(* IEC 61131-3 sources: mect_apps/TP1043_CAN/CANopenClient_PLC, 8 files *)

(* ---- CANopenClient_CAN.gvl ---- *)
(* Global var file *)
VAR_GLOBAL
	ch1_CAN1_IN_DIG_8_1 AT %IB3.4096: BYTE;
	ch1_CAN1_IN_DIG_8_1_1 AT %IX3.4096.0: BOOL;
	ch1_CAN1_IN_DIG_8_1_2 AT %IX3.4096.1: BOOL;
	ch1_CAN1_IN_DIG_8_1_3 AT %IX3.4096.2: BOOL;
	ch1_CAN1_IN_DIG_8_1_4 AT %IX3.4096.3: BOOL;
	ch1_CAN1_IN_DIG_8_1_5 AT %IX3.4096.4: BOOL;
	ch1_CAN1_IN_DIG_8_1_6 AT %IX3.4096.5: BOOL;
	ch1_CAN1_IN_DIG_8_1_7 AT %IX3.4096.6: BOOL;
	ch1_CAN1_IN_DIG_8_1_8 AT %IX3.4096.7: BOOL;

	ch1_CAN1_IN_DIG_8_2 AT %IB3.4097: BYTE;

	ch1_CAN1_OUT_DIG_8_1 AT %QB3.4096: BYTE;
	ch1_CAN1_OUT_DIG_8_1_1 AT %QX3.4096.0: BOOL;
	ch1_CAN1_OUT_DIG_8_1_2 AT %QX3.4096.1: BOOL;
	ch1_CAN1_OUT_DIG_8_1_3 AT %QX3.4096.2: BOOL;
	ch1_CAN1_OUT_DIG_8_1_4 AT %QX3.4096.3: BOOL;
	ch1_CAN1_OUT_DIG_8_1_5 AT %QX3.4096.4: BOOL;
	ch1_CAN1_OUT_DIG_8_1_6 AT %QX3.4096.5: BOOL;
	ch1_CAN1_OUT_DIG_8_1_7 AT %QX3.4096.6: BOOL;
	ch1_CAN1_OUT_DIG_8_1_8 AT %QX3.4096.7: BOOL;

	ch1_CAN1_OUT_DIG_8_2 AT %QB3.4097: BYTE;
	ch1_CAN1_IN_AN_1 AT %IW3.8192: INT;
	ch1_CAN1_IN_AN_2 AT %IW3.8194: INT;
	ch1_3 AT %IW3.8196: INT;
	ch1_4 AT %IW3.8198: INT;
	ch1_5 AT %IW3.8200: INT;
	ch1_6 AT %IW3.8202: INT;
	ch1_CAN1_OUT_AN_1 AT %QW3.8192: INT;
	PLC_CAN1_IN_DIG_8_1 AT %MB0.5380: BYTE;
	PLC_CAN1_IN_DIG_8_2 AT %MB0.5384: BYTE;
	PLC_CAN1_OUT_DIG_8_1 AT %MB0.5388: BYTE;
	PLC_CAN1_OUT_DIG_8_2 AT %MB0.5392: BYTE;
	PLC_CAN1_IN_AN_1 AT %MW0.5396: INT;
	PLC_CAN1_IN_AN_2 AT %MW0.5400: INT;
	PLC_3 AT %MW0.5404: INT;
	PLC_4 AT %MW0.5408: INT;
	PLC_5 AT %MW0.5412: INT;
	PLC_6 AT %MW0.5416: INT;
	PLC_CAN1_OUT_AN_1 AT %MW0.5420: INT;
END_VAR

(* ---- Resource1.gvl ---- *)
(* Global variable file *)
VAR_GLOBAL
DigitalInput_3 AT %MW0.5380:UINT;
DigitalInput_4 AT %MW0.5384:UINT;
DigitalOutput_1 AT %MW0.5388:UINT;
DigitalOutput_2 AT %MW0.5392:UINT;
AnalogInput_1 AT %MW0.5396:INT;
AnalogInput_2 AT %MW0.5400:INT;
END_VAR

(* ---- fb_HW119_AlarmsMngr.st ---- *)
(*[[
]]*)
FUNCTION_BLOCK fb_HW119_AlarmsMngr
#import "Resource1.gvl"
#import "crosstable.gvl"
VAR_INPUT
END_VAR
VAR
	Index:DINT;			(* indice di scansione della CT degli allarmi	*)
	SourceAddr:INT;		(* indirizzo della variabile sorgente	*)
	CompareAdddr:INT;	(* indirizzo della variabile di confronto	*)
	CompareVal:DWORD;	(* valore di confronto	*)
	TagAddr:INT;		(* indirizzo della variabile di allarme	*)
	ERRFlag:BOOL;		(* flag d segnalazione errore nell'esecuzioe di una funzione	*)
	ERRORVAL:DWORD:=16#00000001;	(* *)
	tmp:DWORD;			(* variabile di appoggio	*)
	tmpOld:DWORD;		(* variabile di appoggio	*)
END_VAR
(*
	Blocco funzione per la gestione degli alalrmi/eventi

*)

	IF Index < DimAlarmsCT AND ALCrossTable[Index].ALTag <> '' THEN
		SourceAddr:=WORD_TO_INT(HW119_GetAddr(ALCrossTable[Index].ALSource));		(* ricava l'indirizzo della varibile sorgente*)
		IF SourceAddr = WORD_TO_INT(16#FFFF)  OR SourceAddr > DINT_TO_INT(DimCrossTable) OR SourceAddr = 0  THEN									(* controlla il risultato della funzione*)
			ERRFlag:=TRUE;
		ELSE
			IF	CrossTable[SourceAddr].Error > 0 AND CrossTable[SourceAddr].Protocol<>100 THEN			(* verifica che il valore sia stato aggiornato	*)
				ERRFlag:=TRUE;
			ELSE
				CompareAdddr:=-1;
				IF ALCrossTable[Index].ALCompareVar = '' THEN
					CompareVal:=ALCrossTable[Index].ALCompareVaL;					(* variabile di confronto nulla -> rileva il valore di confronto*)
				ELSE
					CompareAdddr:=WORD_TO_INT(HW119_GetAddr(ALCrossTable[Index].ALCompareVar));	(* ricava l'indirizzo della varibile di confronto *)

					IF CompareAdddr = WORD_TO_INT(16#FFFF) OR CompareAdddr > DINT_TO_INT(DimCrossTable) OR CompareAdddr = 0 THEN					(* controlla se la variable di controllo corretta*)
						ERRFlag:=TRUE;
					ELSE
						IF CrossTable[CompareAdddr].Error > 0 AND CrossTable[CompareAdddr].Protocol<>100 THEN	(* verifica  se la variabile di controllo è nella CT*)
							ERRFlag:=TRUE;
						ELSE
							CompareVal:=ARRAY_CROSSTABLE_INPUT[CompareAdddr];
						END_IF;
					END_IF;
				END_IF;
				TagAddr:=WORD_TO_INT(HW119_GetAddr(ALCrossTable[Index].ALTag));		(* ricavo l'indirizzo della varibile destinazione*)
				IF TagAddr = WORD_TO_INT(16#FFFF) OR TagAddr > DINT_TO_INT(DimCrossTable) OR TagAddr = 0 THEN
					ERRFlag:=TRUE;
				END_IF;
			END_IF;
		END_IF;

		IF NOT ERRFlag	THEN						(* Se i valori letti da CT sono corenti effettua il check di allarme	*)
			tmp:=UINT_TO_DWORD(ALCrossTable[Index].ALOperator)	AND 16#FF00	;	(* controlla l'operazione da eseguire *)
			CASE DWORD_TO_INT(tmp) OF
(*  operatore >	*)		16#100 :
							IF ARRAY_CROSSTABLE_INPUT[SourceAddr] > CompareVal	 THEN
								IF  ALCrossTable[Index].ALFilterCount=0  THEN
									ARRAY_CROSSTABLE_INPUT[TagAddr]:=ERRORVAL;
								ELSE
									ALCrossTable[Index].ALFilterCount:=ALCrossTable[Index].ALFilterCount-1;
								END_IF;
							ELSE
								ARRAY_CROSSTABLE_INPUT[TagAddr]:=0;
								ALCrossTable[Index].ALFilterCount:=ALCrossTable[Index].ALFilterTime;
							END_IF;
(*  operatore >=	*)	16#200 :
							IF ARRAY_CROSSTABLE_INPUT[SourceAddr] >= CompareVal	 THEN
								IF  ALCrossTable[Index].ALFilterCount=0  THEN
									ARRAY_CROSSTABLE_INPUT[TagAddr]:=ERRORVAL;
								ELSE
									ALCrossTable[Index].ALFilterCount:=ALCrossTable[Index].ALFilterCount-1;
								END_IF;
							ELSE
								ARRAY_CROSSTABLE_INPUT[TagAddr]:=0;

							END_IF;
(*  operatore <	*)		16#300 :
							IF ARRAY_CROSSTABLE_INPUT[SourceAddr] < CompareVal	 THEN
								IF  ALCrossTable[Index].ALFilterCount=0  THEN
									ARRAY_CROSSTABLE_INPUT[TagAddr]:=ERRORVAL;

								ELSE
									ALCrossTable[Index].ALFilterCount:=ALCrossTable[Index].ALFilterCount-1;
								END_IF;
							ELSE
								ARRAY_CROSSTABLE_INPUT[TagAddr]:=0;
								ALCrossTable[Index].ALFilterCount:=ALCrossTable[Index].ALFilterTime;
							END_IF;
(*  operatore <=	*)	16#400 :
							IF ARRAY_CROSSTABLE_INPUT[SourceAddr] <= CompareVal	 THEN
								IF  ALCrossTable[Index].ALFilterCount=0  THEN
									ARRAY_CROSSTABLE_INPUT[TagAddr]:=ERRORVAL;

								ELSE
									ALCrossTable[Index].ALFilterCount:=ALCrossTable[Index].ALFilterCount-1;
								END_IF;
							ELSE
								ARRAY_CROSSTABLE_INPUT[TagAddr]:=0;
								ALCrossTable[Index].ALFilterCount:=ALCrossTable[Index].ALFilterTime;
							END_IF;
(*  operatore =	*)		16#500 :
							IF ARRAY_CROSSTABLE_INPUT[SourceAddr] = CompareVal	 THEN
								IF  ALCrossTable[Index].ALFilterCount=0  THEN
									ARRAY_CROSSTABLE_INPUT[TagAddr]:=ERRORVAL;

								ELSE
									ALCrossTable[Index].ALFilterCount:=ALCrossTable[Index].ALFilterCount-1;
								END_IF;
							ELSE
								ARRAY_CROSSTABLE_INPUT[TagAddr]:=0;
								ALCrossTable[Index].ALFilterCount:=ALCrossTable[Index].ALFilterTime;
							END_IF;
(*  operatore <>	*)	16#600 :
							IF ARRAY_CROSSTABLE_INPUT[SourceAddr] <> CompareVal	 THEN
								IF  ALCrossTable[Index].ALFilterCount=0  THEN
									ARRAY_CROSSTABLE_INPUT[TagAddr]:=ERRORVAL;

								ELSE
									ALCrossTable[Index].ALFilterCount:=ALCrossTable[Index].ALFilterCount-1;
								END_IF;
							ELSE
								ARRAY_CROSSTABLE_INPUT[TagAddr]:=0;
								ALCrossTable[Index].ALFilterCount:=ALCrossTable[Index].ALFilterTime;
							END_IF;

						ELSE
(*controllo a bit *)

							tmp:= SHR(ARRAY_CROSSTABLE_INPUT[SourceAddr], WORD_TO_INT ( UINT_TO_WORD ( ALCrossTable[Index].ALOperator) AND 16#00FF)-1 );
							tmp:=tmp AND 16#1;
							(*controllo a bit sui livelli*)

							IF CompareAdddr = -1 THEN

								IF tmp = CompareVal	THEN
									IF  ALCrossTable[Index].ALFilterCount=0  THEN
										ARRAY_CROSSTABLE_INPUT[TagAddr]:=ERRORVAL;

									ELSE
										ALCrossTable[Index].ALFilterCount:=ALCrossTable[Index].ALFilterCount-1;
									END_IF;
								ELSE
									ARRAY_CROSSTABLE_INPUT[TagAddr]:=0;
									ALCrossTable[Index].ALFilterCount:=ALCrossTable[Index].ALFilterTime;
								END_IF;
(* controllo  transizioni*)
							ELSIF CompareAdddr=SourceAddr 	THEN
(* allarme su fronte di salita*)
								tmpOld:= SHR(CrossTable[SourceAddr].OldVal, WORD_TO_INT ( UINT_TO_WORD ( ALCrossTable[Index].ALOperator) AND 16#00FF)-1 );
								tmpOld:=tmpOld AND 16#1;
								IF		tmp = 16#01 AND 	tmpOld=16#00 AND ALCrossTable[Index].ALCompareVal =  FRONTE_SALITA	THEN
								 	ARRAY_CROSSTABLE_INPUT[TagAddr]:=ERRORVAL;
(* allarme su fronte di discesa*)
								ELSIF	tmp = 16#00  AND 	tmpOld=16#01 AND ALCrossTable[Index].ALCompareVal =  FRONTE_DISCESA	THEN
								 	ARRAY_CROSSTABLE_INPUT[TagAddr]:=ERRORVAL;
								ELSIF ALCrossTable[Index].ALCompareVal =  FRONTE_SALITA AND tmp=16#00 THEN
									ARRAY_CROSSTABLE_INPUT[TagAddr]:=0;
								ELSIF ALCrossTable[Index].ALCompareVal =  FRONTE_DISCESA AND tmp= 16#01 THEN
									ARRAY_CROSSTABLE_INPUT[TagAddr]:=0;
								END_IF;
								IF tmp = 0 THEN
									tmp:=16#FFFFFFFE;
									CrossTable[SourceAddr].OldVal:=CrossTable[SourceAddr].OldVal AND ROL(tmp, WORD_TO_INT ( UINT_TO_WORD ( ALCrossTable[Index].ALOperator) AND 16#00FF)-1 );
								ELSE
									CrossTable[SourceAddr].OldVal:=CrossTable[SourceAddr].OldVal OR ROL(tmp, WORD_TO_INT ( UINT_TO_WORD ( ALCrossTable[Index].ALOperator) AND 16#00FF)-1 );
								END_IF;
							END_IF;

			END_CASE;
		END_IF;
		Index:=Index+1;
		ERRFlag:=FALSE;
	ELSE
		Index:=1;
	END_IF;

END_FUNCTION_BLOCK

(* ---- fb_HW119_MODBUS.st ---- *)
(*[[
]]*)
FUNCTION_BLOCK fb_HW119_MODBUS
#import "Resource1.gvl"
#import "crosstable.gvl"
VAR_INPUT
	RdWr:WORD;
	address:INT;
	Index:int;
	Protocol:STRING;
END_VAR
VAR_OUTPUT
	Error:UINT;
END_VAR
VAR
	FunctRes:UINT;
	HeadAddr:INT;
	I:INT;
	STEPS:INT;
	RW:WORD;
	COUNT_ERR:UDINT:=0;
	addr:INT;
	COUNT_CICLI:UDINT;
	regs:INT;
	LowByte:BYTE;
	BOOL_Data:	ARRAY[0..259]	OF BYTE;
	INT_Data:	ARRAY[0..259]	OF UINT;
	tempo1:TIME;
	tempo2:TIME;
	Index_A:int;
	tmpARRAY_CROSSTABLE_OUTPUT:	ARRAY[0..19] OF DWORD;
END_VAR

	tempo1:=TIM_Get();
(*	TRIGGER02:=1;
	TRIGGER01:=1;
	*)

		RW:=RdWr;
		HeadAddr:=address;
		addr:=address;
		Index_A:=Index;

		IF RW > 0   THEN											(* Variabile abilitata*)

			COUNT_CICLI:=COUNT_CICLI+1;
			FunctRes:= MODBUS_SET_SLAVE(Protocol,CrossTable[HeadAddr].NodeId);
			IF FunctRes = 0  THEN										(* Funzione andata a buon fine*)
				MODBUS_ERR[10]:=2;
				IF RW = READ	THEN									(* OPERAZIONE DI LETTURA	*)
					TRIGGER02:=1;
					regs:=0;
					IF Index_A > 0 THEN
						ARRAY_QUEUE_OUTPUT[Index_A]:=STATO_BUSY_READ;	(* metto busy read l'intero blocco*)
					END_IF;
					FOR I:=0 TO CrossTable[HeadAddr].NReg-1 DO				(*  calcolo del numero di letture modbus da effettuare*)

						CASE CrossTable[HeadAddr+I].Types OF
							FLOATABCD,UDINTABCD,DINTABCD:		regs:=regs+2;
							FLOATDCBA,UDINTDCBA,DINTDCBA:		regs:=regs+2;
							FLOATCDAB,UDINTCDAB,DINTCDAB:		regs:=regs+2;
							FLOATBADC,UDINTBADC,DINTBADC:		regs:=regs+2;
						ELSE
							regs:=regs+1;
						END_CASE;
				   	END_FOR;
					IF CrossTable[HeadAddr].Types = BIT THEN			(* richiesta di lettura a bit	*)
						FunctRes:=  MODBUS_READ_BITS (Protocol,CrossTable[HeadAddr].Address,INT_TO_UINT(regs),BOOL_Data);
					ELSE
						FunctRes:= MODBUS_READ_REGISTERS (Protocol,CrossTable[HeadAddr].Address,INT_TO_UINT(regs),INT_Data);
					END_IF;
					IF FunctRes = 0  THEN								(* Funzione andata a buon fine*)
						Error:=0;
						MODBUS_ERR[11]:=2;
						ErrorsState:=ErrorsState AND 16#FF7F;
						CrossTable[HeadAddr].Error:=0;						(* segnala valore valido	*)
						I:=0;
						REPEAT
							CASE CrossTable[HeadAddr].Types OF
								FLOATABCD,UDINTABCD,DINTABCD :		STEPS:=2;
								FLOATDCBA,UDINTDCBA,DINTDCBA:		STEPS:=2;
								FLOATCDAB,UDINTCDAB,DINTCDAB:		STEPS:=2;
								FLOATBADC,UDINTBADC,DINTBADC:		STEPS:=2;
							ELSE
								STEPS:=1;
							END_CASE;
							CASE CrossTable[addr].Types	OF				(* in funzione del tipo di dato sistema la variabile	*)
								FLOATABCD,UDINTABCD,DINTABCD:
									ARRAY_CROSSTABLE_INPUT[addr]:=0;
									ARRAY_CROSSTABLE_INPUT[addr]:=UINT_TO_DWORD(INT_Data[I]) OR SHL(UINT_TO_DWORD(INT_Data[I+1]),16) ;
							(*		DummyFloat:=DWORD_TO_REAL(ARRAY_CROSSTABLE_INPUT[addr+I]);*)

								FLOATDCBA,UDINTDCBA,DINTDCBA:
									ARRAY_CROSSTABLE_INPUT[addr]:=0;
									LowByte:=UINT_TO_BYTE(INT_Data[I]);
									INT_Data[I]:= WORD_TO_UINT(SHR(UINT_TO_WORD(INT_Data[I]),8));
									INT_Data[I]:=	WORD_TO_UINT(UINT_TO_WORD(INT_Data[I]) OR  SHL(BYTE_TO_WORD(LowByte),8));
									LowByte:=UINT_TO_BYTE(INT_Data[I+1]);
									INT_Data[I+1]:= WORD_TO_UINT(SHR(UINT_TO_WORD(INT_Data[I+1]),8));
									INT_Data[I+1]:=	WORD_TO_UINT(UINT_TO_WORD(INT_Data[I+1]) OR  SHL(BYTE_TO_WORD(LowByte),8));
									ARRAY_CROSSTABLE_INPUT[addr]:=UINT_TO_DWORD(INT_Data[I+1]) OR SHL(UINT_TO_DWORD(INT_Data[I]),16) ;

								FLOATCDAB,UDINTCDAB,DINTCDAB:
									ARRAY_CROSSTABLE_INPUT[addr]:=0;
									ARRAY_CROSSTABLE_INPUT[addr]:=UINT_TO_DWORD(INT_Data[I+1]) OR SHL(UINT_TO_DWORD(INT_Data[I]),16) ;

								FLOATBADC,UDINTBADC,DINTBADC:
									ARRAY_CROSSTABLE_INPUT[addr]:=0;
									LowByte:=UINT_TO_BYTE(INT_Data[I]);
									INT_Data[I]:= WORD_TO_UINT(SHR(UINT_TO_WORD(INT_Data[I]),8));
									INT_Data[I]:=	WORD_TO_UINT(UINT_TO_WORD(INT_Data[I]) OR  SHL(BYTE_TO_WORD(LowByte),8));
									LowByte:=UINT_TO_BYTE(INT_Data[I+1]);
									INT_Data[I+1]:= WORD_TO_UINT(SHR(UINT_TO_WORD(INT_Data[I+1]),8));
									INT_Data[I+1]:=	WORD_TO_UINT(UINT_TO_WORD(INT_Data[I+1]) OR  SHL(BYTE_TO_WORD(LowByte),8));
									ARRAY_CROSSTABLE_INPUT[addr]:=UINT_TO_DWORD(INT_Data[I]) OR SHL(UINT_TO_DWORD(INT_Data[I+1]),16) ;
								UINT16:
									ARRAY_CROSSTABLE_INPUT[addr]:=UINT_TO_DWORD(INT_Data[I]);
								INT16:
									ARRAY_CROSSTABLE_INPUT[addr]:=UINT_TO_DWORD(INT_Data[I]);
								BIT:
									ARRAY_CROSSTABLE_INPUT[addr]:=BYTE_TO_DWORD(BOOL_Data[I]);
							ELSE
								ARRAY_CROSSTABLE_INPUT[addr]:=UINT_TO_DWORD(INT_Data[I]);
							END_CASE;
							addr:=addr+1;							(* punta alla successiva variabile della crosstable*)
							I:=I+STEPS;
						UNTIL I >= regs
						END_REPEAT;
						FOR I:=0 TO CrossTable[HeadAddr].NReg-1	DO
							ARRAY_STATES[HeadAddr+I]:=STATO_OK;				(* segnala lo stato della comunicazione a OK		*)
							CrossTable[HeadAddr+I].Error:=0;						(* segnala valore valido	*)
						END_FOR;
					ELSIF FunctRes > 0	THEN						(*	segnala lo stato della comunicazione a  ERR		*)
						MODBUS_ERR[11]:=3;
						ErrorsState:=ErrorsState OR 16#0080;
						Error:=FunctRes;
						FOR I:=0 TO CrossTable[HeadAddr].NReg-1	DO
							ARRAY_STATES[HeadAddr+I]:=STATO_ERR;
							CrossTable[HeadAddr+I].Error:=1;					(* segnala valore non valido *)
						END_FOR;
						COUNT_ERR:=COUNT_ERR+1;
					END_IF;
				ELSIF  RW =  WRITE_SINGLE OR RW = WRITE_MULTIPLE OR RW = WRITE_RIC_SINGLE  OR RW = WRITE_RIC_MULTIPLE    THEN												(*	OPERAZIONE DI SCRITTURA	*)
					regs:=0;
					RW:=RW AND 16#B000;
					IF RW=WRITE_SINGLE THEN							(* scrittura singola ingnoro il contenuto di Nreg*)
						IF Index_A > 0 THEN
							ARRAY_QUEUE_OUTPUT[Index_A]:=STATO_BUSY_WRITE;
							tmpARRAY_CROSSTABLE_OUTPUT[0]:=ARRAY_CROSSTABLE_OUTPUT[HeadAddr];
						ELSE
							tmpARRAY_CROSSTABLE_OUTPUT[0]:=CrossTable[HeadAddr].PLCWriteVal;
						END_IF;
						ARRAY_STATES[HeadAddr]:=STATO_RUN;
						CASE CrossTable[HeadAddr].Types OF
							FLOATABCD,UDINTABCD,DINTABCD:		regs:=2;
							FLOATDCBA,UDINTDCBA,DINTDCBA:		regs:=2;
							FLOATCDAB,UDINTCDAB,DINTCDAB:		regs:=2;
							FLOATBADC,UDINTBADC,DINTBADC:		regs:=2;
						ELSE
							regs:=1;
						END_CASE;

					ELSIF RW = WRITE_MULTIPLE THEN
						IF Index_A > 0 THEN
							ARRAY_QUEUE_OUTPUT[Index_A]:=STATO_BUSY_WRITE;
						END_IF;

						FOR I:=0 TO CrossTable[HeadAddr].NReg-1 DO				(*  calcolo del numero di letture modbus da effettuare*)
							IF Index_A > 0 THEN
								tmpARRAY_CROSSTABLE_OUTPUT[I]:=ARRAY_CROSSTABLE_OUTPUT[HeadAddr+I];
							ELSE
								tmpARRAY_CROSSTABLE_OUTPUT[I]:=CrossTable[HeadAddr+I].PLCWriteVal;
							END_IF;

							ARRAY_STATES[HeadAddr+I]:=STATO_RUN;
							CASE CrossTable[HeadAddr+I].Types OF
								FLOATABCD,UDINTABCD,DINTABCD:		regs:=regs+2;
								FLOATDCBA,UDINTDCBA,DINTDCBA:		regs:=regs+2;
								FLOATCDAB,UDINTCDAB,DINTCDAB:		regs:=regs+2;
								FLOATBADC,UDINTBADC,DINTBADC:		regs:=regs+2;
							ELSE
								regs:=regs+1;
							END_CASE;
					   	END_FOR;
					END_IF;

					I:=0;
					REPEAT
						CASE CrossTable[addr].Types OF
							FLOATABCD,UDINTABCD,DINTABCD :		STEPS:=2;
							FLOATDCBA,UDINTDCBA,DINTDCBA:		STEPS:=2;
							FLOATCDAB,UDINTCDAB,DINTCDAB:		STEPS:=2;
							FLOATBADC,UDINTBADC,DINTBADC:		STEPS:=2;
						ELSE
							STEPS:=1;
						END_CASE;

						CASE CrossTable[addr].Types	OF				(* in funzione del tipo di dato arrangia la variabile	*)

							FLOATDCBA,UDINTDCBA,DINTDCBA:
								INT_Data[I+1]:=DWORD_TO_UINT(tmpARRAY_CROSSTABLE_OUTPUT[addr-HeadAddr] AND 16#0000FFFF);
								INT_Data[I]:=DWORD_TO_UINT(SHR(tmpARRAY_CROSSTABLE_OUTPUT[addr-HeadAddr],16) AND 16#0000FFFF);
								LowByte:=UINT_TO_BYTE(INT_Data[I]);
								INT_Data[I]:= WORD_TO_UINT(SHR(UINT_TO_WORD(INT_Data[I]),8));
								INT_Data[I]:=	WORD_TO_UINT(UINT_TO_WORD(INT_Data[I]) OR  SHL(BYTE_TO_WORD(LowByte),8));
								LowByte:=UINT_TO_BYTE(INT_Data[I+1]);
								INT_Data[I+1]:= WORD_TO_UINT(SHL(UINT_TO_WORD(INT_Data[I+1]),8));
								INT_Data[I+1]:=	WORD_TO_UINT(UINT_TO_WORD(INT_Data[I+1]) OR  SHL(BYTE_TO_WORD(LowByte),8));

							FLOATCDAB,UDINTCDAB,DINTCDAB:
								INT_Data[I+1]:=DWORD_TO_UINT(tmpARRAY_CROSSTABLE_OUTPUT[addr-HeadAddr] AND 16#0000FFFF);
								INT_Data[I]:=DWORD_TO_UINT(SHL(tmpARRAY_CROSSTABLE_OUTPUT[addr-HeadAddr],16) AND 16#0000FFFF);

							FLOATBADC,UDINTBADC,DINTBADC:
								INT_Data[I]:=DWORD_TO_UINT(tmpARRAY_CROSSTABLE_OUTPUT[addr-HeadAddr] AND 16#0000FFFF);
								INT_Data[I+1]:=DWORD_TO_UINT(SHR(tmpARRAY_CROSSTABLE_OUTPUT[addr-HeadAddr],16) AND 16#0000FFFF);
								LowByte:=UINT_TO_BYTE(INT_Data[I]);
								INT_Data[I]:= WORD_TO_UINT(SHR(UINT_TO_WORD(INT_Data[I]),8));
								INT_Data[I]:=	WORD_TO_UINT(UINT_TO_WORD(INT_Data[I]) OR  SHL(BYTE_TO_WORD(LowByte),8));
								LowByte:=UINT_TO_BYTE(INT_Data[I+1]);
								INT_Data[I+1]:= WORD_TO_UINT(SHL(UINT_TO_WORD(INT_Data[I+1]),8));
								INT_Data[I+1]:=	WORD_TO_UINT(UINT_TO_WORD(INT_Data[I+1]) OR  SHL(BYTE_TO_WORD(LowByte),8));

							UINT16:	INT_Data[I]:=DWORD_TO_UINT(tmpARRAY_CROSSTABLE_OUTPUT[addr-HeadAddr] AND 16#0000FFFF);

							INT16:	INT_Data[I]:=DWORD_TO_UINT(tmpARRAY_CROSSTABLE_OUTPUT[addr-HeadAddr] AND 16#0000FFFF);

							BIT:	BOOL_Data[I]:=DWORD_TO_BYTE(tmpARRAY_CROSSTABLE_OUTPUT[addr-HeadAddr] AND 16#0000FFFF);

						ELSE
							INT_Data[I]:=DWORD_TO_UINT(tmpARRAY_CROSSTABLE_OUTPUT[addr-HeadAddr] AND 16#0000FFFF);
							INT_Data[I+1]:=DWORD_TO_UINT(SHR(tmpARRAY_CROSSTABLE_OUTPUT[addr-HeadAddr],16) AND 16#0000FFFF);

						END_CASE;
						I:=I+STEPS;
						addr:=addr+1;							(* punta alla successiva variabile della crosstable*)

					UNTIL I >= regs
				    END_REPEAT;

					IF  CrossTable[HeadAddr].Types = BIT	THEN		(* richiesta scrittura a bit*)
						FunctRes:= MODBUS_WRITE_BITS (Protocol,CrossTable[HeadAddr].Address,INT_TO_UINT(regs),BOOL_Data);
					ELSE												(*riciesta scrittura a word*)
						IF regs = 1	THEN
							FunctRes:= MODBUS_WRITE_REGISTER (Protocol,CrossTable[HeadAddr].Address,INT_Data[0]);
						ELSE
							FunctRes:= MODBUS_WRITE_REGISTERS (Protocol,CrossTable[HeadAddr].Address,regs,INT_Data);
						END_IF;
					END_IF;
					IF FunctRes = 0  THEN							(*	Funzione andata a buon fine *)
						MODBUS_ERR[12]:=2;
						ErrorsState:=ErrorsState AND 16#FF7F;
						IF RW=WRITE_SINGLE THEN
							IF Index_A > 0	THEN
								ARRAY_CROSSTABLE_INPUT[HeadAddr]:=ARRAY_CROSSTABLE_OUTPUT[HeadAddr];
							ELSE
								ARRAY_CROSSTABLE_INPUT[HeadAddr]:=CrossTable[HeadAddr].PLCWriteVal;
							END_IF;
							ARRAY_STATES[HeadAddr]:=STATO_OK;				(* segnala lo stato della comunicazione a OK		*)
						ELSE

							FOR I:=0 TO  CrossTable[HeadAddr].NReg-1 DO			(*	copia dei valori da leggere nel buffer di comunicazione	*)
								IF Index_A > 0	THEN
									ARRAY_CROSSTABLE_INPUT[HeadAddr+I]:=ARRAY_CROSSTABLE_OUTPUT[HeadAddr+I];
								ELSE
									ARRAY_CROSSTABLE_INPUT[HeadAddr+I]:=CrossTable[HeadAddr+I].PLCWriteVal;
								END_IF;
								ARRAY_STATES[HeadAddr+I]:=STATO_OK;				(* segnala lo stato della comunicazione a OK		*)

							END_FOR;
						END_IF;
						Error:=0;
					ELSIF FunctRes > 0	THEN
						Error:=FunctRes;
						MODBUS_ERR[12]:=3;
						COUNT_ERR:=COUNT_ERR+1;
						ErrorsState:=ErrorsState OR 16#0080;
						IF RW = WRITE_SINGLE THEN
							ARRAY_STATES[HeadAddr]:=STATO_ERR;
						ELSE
							FOR I:=0 TO  CrossTable[HeadAddr].NReg-1 DO
								ARRAY_STATES[HeadAddr+I]:=STATO_ERR;
							END_FOR;
						END_IF;
					END_IF;

				END_IF;
			ELSE
				MODBUS_ERR[10]:=3;
			END_IF;
	 	END_IF;
	tempo2:=TIM_Get()-tempo1;

END_FUNCTION_BLOCK

(* ---- fb_HW119_PLCwriteVar.st ---- *)
(*[[
]]*)
FUNCTION_BLOCK fb_HW119_PLCwriteVar
#import "Resource1.gvl"
#import "crosstable.gvl"
VAR_INPUT
	VARIABLE:STRING;		(* Mnemonico della variabile da scrivere	*)
	VALUES: ARRAY [0..15] OF DWORD;			(* valori da scrivere		*)
	Nregs:INT;
END_VAR
VAR_OUTPUT
	ERR:BOOL;				(* Segnala un errore nell'esecuzione del blocco funzione	*)
END_VAR
VAR
	ADDRESS:WORD;
	I:INT;
	tempo1:TIME;
END_VAR
(*
	Blocco funzione per la scrittura di una variabile attraverso  il PLC di controllo

*)
	ERR:=FALSE;
	ADDRESS:=HW119_GetAddr(VARIABLE);
	tempo1:=TIM_Get();

		IF ADDRESS = 16#FFFF 	THEN
			ERR:=TRUE;
		ELSE
			FOR I:=0 TO NRegs-1 DO											(*  calcolo del numero di scritture modbus da effettuare*)
				CrossTable[WORD_TO_INT(ADDRESS)+I].PLCWriteVal:=VALUES[I];
			END_FOR;
			CASE 	CrossTable[WORD_TO_INT(ADDRESS)].Protocol OF

				0:	IF RTUProtocol_ON THEN
						LocalRTUQueue[IndexRTUQueuePut]:=ADDRESS;
						RTURequestPLCWrite:=RTURequestPLCWrite+1;
						IndexRTUQueuePut:=IndexRTUQueuePut+1;
						if IndexRTUQueuePut > MaxLocalQueue then
							IndexRTUQueuePut:=0;
						end_if;
						CrossTable[WORD_TO_INT(ADDRESS)].Counter:=Nregs;
					END_IF;

				1:	IF TCPProtocol_ON THEN
						LocalTCPQueue[IndexTCPQueuePut]:=ADDRESS;
						TCPRequestPLCWrite:=TCPRequestPLCWrite+1;
						IndexTCPQueuePut:=IndexTCPQueuePut+1;
						if IndexTCPQueuePut > MaxLocalQueue then
							IndexTCPQueuePut:=0;
						end_if;
						CrossTable[WORD_TO_INT(ADDRESS)].Counter:=Nregs;
					END_IF;
				2:	IF TCPRTUProtocol_ON 	THEN
						LocalTCPRTUQueue[IndexTCPRTUQueuePut]:=ADDRESS;
						TCPRTURequestPLCWrite:=TCPRTURequestPLCWrite+1;
						IndexTCPRTUQueuePut:=IndexTCPRTUQueuePut+1;
						if IndexTCPRTUQueuePut > MaxLocalQueue then
							IndexTCPRTUQueuePut:=0;
						end_if;
						CrossTable[WORD_TO_INT(ADDRESS)].Counter:=Nregs;
					END_IF;
				ELSE
					FOR I:=0 TO NRegs-1 DO											(* aggiorno l'array di input con le variabili da scrivere*)
						ARRAY_CROSSTABLE_INPUT[WORD_TO_INT(ADDRESS)+I]:=CrossTable[WORD_TO_INT(ADDRESS)+I].PLCWriteVal;
						CrossTable[WORD_TO_INT(ADDRESS)+I].Error:=0;
					END_FOR;
					TRIGGER01:=1;
			END_CASE;
		END_IF;

END_FUNCTION_BLOCK

(* ---- fb_HW119_ReadCommFields.st ---- *)
(*[[
]]*)
FUNCTION_BLOCK fb_HW119_ReadCommFields
#import "Resource1.gvl"
#import "crosstable.gvl"
VAR_INPUT
	index:INT;
END_VAR
VAR_OUTPUT
	ERR:BOOL;
END_VAR

VAR
	Field:STRING;
	FunctRes:UINT;
END_VAR

	ERR:=FALSE;
	IF  index = 1 THEN
		FunctRes:=HW119_GetCrossTableField(Field);					(* Number of fails	*)
		IF FunctRes = 0 THEN
			NumberOfFails:=STRING_TO_INT(Field);;
		ELSE
			ERR:=TRUE;
		END_IF;

		FunctRes:=HW119_GetCrossTableField(Field);
		IF FunctRes = 0 THEN										(* Fail  divisor	*)
			FailDivisor:=STRING_TO_BYTE(Field);
		ELSE
			ERR:=TRUE;
		END_IF;
	ELSIF index = 2 THEN

		FunctRes:=HW119_GetCrossTableField(Field);					(* Talta 	*)
		IF FunctRes = 0 THEN
			Talta:=STRING_TO_DINT(Field);
		ELSE
			ERR:=TRUE;
		END_IF;

		FunctRes:=HW119_GetCrossTableField(Field);
		IF FunctRes = 0 THEN										(* Tmedia	*)
			Tmedia:=STRING_TO_DINT(Field);
		ELSE
			ERR:=TRUE;
		END_IF;

		FunctRes:=HW119_GetCrossTableField(Field);
		IF FunctRes = 0 THEN										(* Tbassa	*)
			Tbassa:=STRING_TO_DINT(Field);
		ELSE
			ERR:=TRUE;
		END_IF;

	ELSE

		FunctRes:=HW119_GetCrossTableField(Field);					(* Device	*)
		IF FunctRes = 0 THEN
			CommParameters[index-2].Device:=Field;
		ELSE
			ERR:=TRUE;
		END_IF;

		FunctRes:=HW119_GetCrossTableField(Field);					(* Indirizzo IP	*)
		IF FunctRes = 0 THEN
			CommParameters[index-2].IPaddr:=Field;
		ELSE
			ERR:=TRUE;
		END_IF;

		FunctRes:=HW119_GetCrossTableField(Field);
		IF FunctRes = 0 THEN									(* Port	*)
			CommParameters[index-2].Port:=STRING_TO_UINT(Field);
		ELSE
			ERR:=TRUE;
		END_IF;

		FunctRes:=HW119_GetCrossTableField(Field);					(* Baudrate	*)
		IF FunctRes = 0 THEN
			CommParameters[index-2].BaudRate:=STRING_TO_UINT(Field);
		ELSE
			ERR:=TRUE;
		END_IF;

		FunctRes:=HW119_GetCrossTableField(Field);					(* Parità	*)
		IF FunctRes = 0 THEN
			CommParameters[index-2].Parity:=Field;
		ELSE
			ERR:=TRUE;
		END_IF;

		FunctRes:=HW119_GetCrossTableField(Field);					(* DataBit*)
		IF FunctRes = 0 THEN
			CommParameters[index-2].DataBit:=STRING_TO_UINT(Field);
		ELSE
			ERR:=TRUE;
		END_IF;

		FunctRes:=HW119_GetCrossTableField(Field);					(* StopBit	*)
		IF FunctRes = 0 THEN
			CommParameters[index-2].StopBit:=STRING_TO_UINT(Field);
		ELSE
			ERR:=TRUE;
		END_IF;

		FunctRes:=HW119_GetCrossTableField(Field);					(* Tmin	*)
		IF FunctRes = 0 THEN
			CommParameters[index-2].Tmin:=STRING_TO_INT(Field);
		ELSE
			ERR:=TRUE;
		END_IF;

		FunctRes:=HW119_GetCrossTableField(Field);					(* Timeout	*)
		IF FunctRes = 0 THEN
			CommParameters[index-2].TimeOut:=STRING_TO_UINT(Field);
		ELSE
			ERR:=TRUE;
		END_IF;
	END_IF;

END_FUNCTION_BLOCK

(* ---- PLC.st ---- *)
(*[[
]]*)
PROGRAM PLC
#import "Resource1.gvl"
#import "crosstable.gvl"
#import "CANopenClient_CAN.gvl"
VAR
	info : TSK_INFO ;
	counter : INT := 0;
	task_ms : INT := -1;
	square_ms : INT := 1000;
	retval : WORD;
	first : BOOL := true;
END_VAR;
	if first then
		first := false;
		if task_ms < 0 then
			retval := TSK_GetInfo('Task0_Control', info);
			task_ms := TIME_TO_INT(info.tCycle);
		end_if;
	end_if;

	counter := (counter + 1) mod 10000;

	(* CANopen reading inputs *)
	DigitalInput_3 := BOOL_TO_UINT(ch1_CAN1_IN_DIG_8_1_3);
	DigitalInput_4 := BOOL_TO_UINT(ch1_CAN1_IN_DIG_8_1_4);
	AnalogInput_1 := ch1_CAN1_IN_AN_1;
	AnalogInput_2 := ch1_CAN1_IN_AN_2;

	(* CANopen writing output 1 *)
	if (counter mod (2 * square_ms / task_ms)) < (square_ms / task_ms) then
		DigitalOutput_1 := 1;
	else
		DigitalOutput_1 := 0;
	end_if;
	ch1_CAN1_OUT_DIG_8_1_1 := UINT_TO_BOOL(DigitalOutput_1);

	(* CANopen writing output 2 *)
	DigitalOutput_2 := DigitalInput_4;
	ch1_CAN1_OUT_DIG_8_1_2 := UINT_TO_BOOL(DigitalOutput_2);

END_PROGRAM

(* ---- TCP_Communication.st ---- *)
(*[[
]]*)
PROGRAM TCP_Communication
#import "Resource1.gvl"
#import "crosstable.gvl"
VAR
	HeadAddr:INT;
	ReadWrite:WORD;
	IndexProt_i:ARRAY [0..4] OF INT;
	TON_0:TON;
	TON_1:TON;
	TON_2:TON;
	TON_3:TON;
	BusAccess:fb_HW119_MODBUS;
	FirstCy:BOOL;
	dummy:WORD;
	Enablei: ARRAY [0..3] OF BOOL;
	pointer:INT;
	FlagPrimoCiclo:BOOL;
	Retry:BOOL:=FALSE;
	Protocollo:UINT:=TCP;
	time2:TIME;
	zero:TIME;
	RicettaON:BOOL;
	LastID:INT;
	FirstID:INT;
	I:INT;
	Start:ARRAY [0..4] OF BOOL;
	k:dword;
	j:dword;
END_VAR

TON_0(IN := TRUE,PT := INT_TO_TIME(CommParameters[Protocollo+1].Tmin));
				TON_1(IN := TRUE,PT := DINT_TO_TIME(Talta));
				TON_2(IN := TRUE,PT := DINT_TO_TIME(Tmedia));
				TON_3(IN := TRUE,PT := DINT_TO_TIME(Tbassa));

IF NOT FirstCy THEN
	dummy:=	WD_Disable('Task3_TCP');
	FirstCy:=TRUE;
END_IF;

IF 	TON_0.Q THEN																(* controlla se TIMER Tmin scaduto	*)
	TRIGGER02:=1;
	TRIGGER01:=1;

	TON_0(In:=FALSE);

	IF Reset_TCP =1 THEN
		FOR I:=1 TO 64 DO
			CounterTCP[I]:=0;
		 END_FOR;
		TCPBlackList_ERROR_WORD:=0;
		TCPComm_ERROR_WORD:=0;
		BlackListTCPL:=0;
		BlackListTCPH:=0;
		CommErrTCPL:=0;
		CommErrTCPH:=0;
		ERROR_FLAG:=ERROR_FLAG AND 16#FFFD;

	END_IF;
	IF NOT Retry THEN
		IF TCPRequestPLCWrite > 0 THEN											(* controlla seci sono richieste di scrittura da parte del PLC	*)
			pointer:=4;
			FlagPrimoCiclo:=FALSE;
			IndexProt_i[pointer]:=0;
			HeadAddr:=WORD_TO_INT(LocalRTUQueue[IndexRTUQueueGet]);		(*inizializza i parametri da assegnare al blocco funzione*)
			IF CrossTable[HeadAddr].Counter=1 THEN
				ReadWrite:=WRITE_SINGLE;											(*inizializza i parametri da assegnare al blocco funzione*)
			ELSE
				ReadWrite:=WRITE_MULTIPLE;											(*inizializza i parametri da assegnare al blocco funzione*)
			END_IF;
			TCPRequestPLCWrite:=TCPRequestPLCWrite-1;							(* incrementa il contatore delle scritture effettuate*)
			IndexTCPQueueGet:=IndexTCPQueueGet+1;								(* incrementa il puntatore alla coda *)
			IF IndexTCPQueueGet > MaxLocalQueue THEN
				IndexTCPQueueGet:=0;
			END_IF;
		ELSE
			IF RichiestaScrittura=1 THEN										(* controlla se ci sono richieste di SCRITTURA da parte HMI*)
				IF FlagPrimoCiclo = FALSE THEN									(* controlla se è il primo ingrsso nel ramo a seguito dell'interrupt*)
					FlagPrimoCiclo:=TRUE;										(* Prima richiesta di scrittura => azzero l'indice della coda 	*)
					IndexProt_i[3]:=0;											(* per eseguire le scritture nella sequenza di arrivo		  	*)
					pointer:=3;
					zero:=TIM_Get();
				END_IF;
				REPEAT 															(* Rileva la succssiva variabile a cui accedere nella coda			*)
					IF IndexProt_i[3] < DINT_TO_INT(DimCrossTable) THEN
						IndexProt_i[3]:=IndexProt_i[3]+1;
						ReadWrite:=ARRAY_QUEUE[IndexProt_i[3]] AND QueueRWMask;
						HeadAddr:=WORD_TO_INT(ARRAY_QUEUE[IndexProt_i[3]] AND QueueAddressMask);
						IF HeadAddr < DINT_TO_INT(DimCrossTable) 	THEN
							IF  (ReadWrite = 0  ) OR ( (CrossTable[HeadAddr].Protocol = Protocollo) AND ReadWrite>=WRITE AND (ARRAY_QUEUE_OUTPUT[IndexProt_i[3]]<>STATO_BUSY_WRITE) )   THEN

								IF ReadWrite = 0 THEN
									ARRAY_QUEUE_OUTPUT[IndexProt_i[3]]:=0;
									IF HeadAddr = 0 THEN
										IndexProt_i[3]:=0;
									END_IF;
								ELSIF ReadWrite = WRITE_RIC_SINGLE  OR ReadWrite = WRITE_RIC_MULTIPLE  THEN
									IF NOT RicettaON THEN
										FirstID:=IndexProt_i[3];
										RicettaON:=TRUE;
									END_IF;

									LastID:=IndexProt_i[3];
								END_IF;
								IF ReadWrite>=WRITE THEN
									time2:=TIM_Get()-zero;
								END_IF;

								EXIT;
							END_IF;
						END_IF;
					ELSE
						IndexProt_i[3]:=0;
					END_IF;
				UNTIL  FALSE
				END_REPEAT;
			ELSIF RicettaON AND RichiestaScrittura=0 THEN
				RicettaON:=FALSE;
				FlagPrimoCiclo:=FALSE;
				FOR I:=1 TO  LastID DO
 					ARRAY_QUEUE_OUTPUT[I]:=0;
				END_FOR;
			ELSE																(* richieste di LETTURE	*)
				IF  RichiestaScrittura=0	THEN

					FlagPrimoCiclo:=FALSE;											(* azzera l'akwnoledge dell'interrupt*)
				END_IF;
			END_IF;
			IF  RichiestaScrittura=0	THEN
				IF TON_1.Q OR Enablei[0]=TRUE THEN							(* scaduto il timer ad alta priorità esegue le letture *)
					IF Enablei[0]=FALSE THEN
						TON_1(IN := FALSE);										(* riarma il timer*)
						Start[0]:=TRUE;
					END_IF;
					pointer:=0;
					Enablei[0]:=TRUE;
				ELSIF TON_2.Q OR Enablei[1]=TRUE THEN						(* scaduto il timer ad media priorità esegue le letture *)
					IF Enablei[1]=FALSE THEN
						TON_2(IN := FALSE);										(* riarma il timer*)
						Start[1]:=TRUE;
					END_IF;
					TON_2(IN := FALSE);										(* riarma il timer*)
					pointer:=1;
					Enablei[1]:=TRUE;
				ELSIF TON_3.Q OR Enablei[2]=TRUE THEN						(* scaduto il timer ad media priorità esegue le letture *)
					IF Enablei[2]=FALSE THEN
						TON_3(IN := FALSE);										(* riarma il timer*)
						Start[2]:=TRUE;
					END_IF;
					pointer:=2;
					Enablei[2]:=TRUE;
				END_IF;
		(*		pointer:=0;		*)
				IF Enablei[0] OR Enablei[1] OR Enablei[2] THEN
					REPEAT 															(* Rileva la prima variabile da leggere della cross table*)
						IF IndexProt_i[pointer] < DINT_TO_INT(DimCrossTable) THEN
							IndexProt_i[pointer]:=IndexProt_i[pointer]+1;
							ReadWrite:=ARRAY_QUEUE[IndexProt_i[pointer]] AND QueueRWMask;
							HeadAddr:=WORD_TO_INT(ARRAY_QUEUE[IndexProt_i[pointer]] AND QueueAddressMask);
							IF HeadAddr < DINT_TO_INT(DimCrossTable) 	THEN
								IF ((ReadWrite = 0) OR (CrossTable[HeadAddr].Protocol = Protocollo) AND (CrossTable[HeadAddr].Enable = pointer+1) )    THEN
									IF ReadWrite = 0 THEN
										Enablei[pointer]:=FALSE;
										ARRAY_QUEUE_OUTPUT[IndexProt_i[pointer]]:=0;
										IF HeadAddr = 0 THEN
											IndexProt_i[pointer]:=0;
										END_IF;
									END_IF;
									EXIT;
								END_IF;
							END_IF;
						ELSE
							IndexProt_i[pointer]:=0;
						END_IF;
					UNTIL  FALSE
					END_REPEAT;
				ELSE
					ReadWrite:=0;
				END_IF;

			END_IF;
		END_IF;
	END_IF;
	IF ReadWrite > 0 THEN
		IF Crosstable[HeadAddr].NodeId > 0 AND Crosstable[HeadAddr].NodeId < 64 THEN
			IF TCPListDevices[BYTE_TO_INT(Crosstable[HeadAddr].NodeId)].BlackListed < 2  THEN			(* controlla se il device non è in blacklist*)
				BusAccess(Protocol:='TCP',Index:=IndexProt_i[pointer],address:=HeadAddr,RdWr:=ReadWrite);		(* effettua l'accesso al bus*)
				TON_0(IN := TRUE,PT := INT_TO_TIME(CommParameters[Protocollo+1].Tmin));						(* riarmo di Tmin*)
				IF BusAccess.Error > 0  THEN																(* controlla sec'è stato un errore di comuicazione*)
					ERROR_FLAG:=ERROR_FLAG OR 16#2;
					CounterTCP[BYTE_TO_INT(Crosstable[HeadAddr].NodeId)]:=UDINT_TO_WORD(WORD_TO_UDINT(CounterTCP[BYTE_TO_INT(Crosstable[HeadAddr].NodeId)])+1);
					IF BusAccess.Error = CommError THEN
						TCPComm_ERROR_WORD:=1;
						IF BYTE_TO_INT(Crosstable[HeadAddr].NodeId) > 32 THEN
							CommErrTCPH:=CommErrTCPH OR SHL(16#1,BYTE_TO_INT(Crosstable[HeadAddr].NodeId) -33);
						ELSE
							CommErrTCPL:=CommErrTCPL OR SHL(16#1,BYTE_TO_INT(Crosstable[HeadAddr].NodeId)-1 );
						END_IF;
						Retry:=FALSE;
					ELSIF BusAccess.Error = TimeoutError  THEN		(* controlla se c'è stato un erore di timeout*)
						Retry:=TRUE;							(* imposta il flag retry a TRUE in modo da effettuare le ripetizioni *)
						TCPListDevices[BYTE_TO_INT(Crosstable[HeadAddr].NodeId)].RetryCounter:=TCPListDevices[BYTE_TO_INT(Crosstable[HeadAddr].NodeId)].RetryCounter+1;
						IF TCPListDevices[BYTE_TO_INT(Crosstable[HeadAddr].NodeId)].RetryCounter >= NumberOfFails THEN
							TCPListDevices[BYTE_TO_INT(Crosstable[HeadAddr].NodeId)].BlackListed:=TCPListDevices[BYTE_TO_INT(Crosstable[HeadAddr].NodeId)].BlackListed+1;
							TCPListDevices[BYTE_TO_INT(Crosstable[HeadAddr].NodeId)].JumpRead:=BYTE_TO_INT(FailDivisor);
							Retry:=FALSE;
							IF TCPListDevices[BYTE_TO_INT(Crosstable[HeadAddr].NodeId)].BlackListed > 1 THEN
								TCPBlackList_ERROR_WORD:=1;
								TCP_RUN:=FALSE;
								IF BYTE_TO_INT(Crosstable[HeadAddr].NodeId) > 32 THEN
									BlackListTCPH:=BlackListTCPH OR SHL(16#1,BYTE_TO_INT(Crosstable[HeadAddr].NodeId) -33);
								ELSE
									k:=SHL(16#1,BYTE_TO_INT(Crosstable[HeadAddr].NodeId)-1 );
									BlackListTCPL:=BlackListTCPL OR k;
								END_IF;
							END_IF;
						END_IF;
					END_IF;
				ELSE

					Retry:=FALSE;
					IF BYTE_TO_INT(Crosstable[HeadAddr].NodeId) > 32 THEN
						CommErrTCPH:=CommErrTCPH AND ROL(16#FFFFFFFE,BYTE_TO_INT(Crosstable[HeadAddr].NodeId) -33);
						BlackListTCPH:=BlackListTCPH AND ROL(16#FFFFFFFE,BYTE_TO_INT(Crosstable[HeadAddr].NodeId) -33);
					ELSE
						CommErrTCPL:=CommErrTCPL AND ROL(16#FFFFFFFE,BYTE_TO_INT(Crosstable[HeadAddr].NodeId)-1 );
						k:=ROL(16#FFFFFFFE,BYTE_TO_INT(Crosstable[HeadAddr].NodeId)-1 );
						j:=BlackListTCPL;
						j:=j AND k;
						BlackListTCPL:=j;
					END_IF;
					IF CommErrTCPH =0 AND CommErrTCPl = 0 THEN
						TCPComm_ERROR_WORD:=0;
					END_IF;
					IF BlackListTCPH =0 AND BlackListTCPL = 0 THEN
						TCPBlackList_ERROR_WORD:=0;
					END_IF;

					TCPListDevices[BYTE_TO_INT(Crosstable[HeadAddr].NodeId)].BlackListed:=0;
					TCPListDevices[BYTE_TO_INT(Crosstable[HeadAddr].NodeId)].RetryCounter:=0;
				END_IF;
			ELSE
				TCPListDevices[BYTE_TO_INT(Crosstable[HeadAddr].NodeId)].JumpRead:=TCPListDevices[BYTE_TO_INT(Crosstable[HeadAddr].NodeId)].JumpRead-1;
				IF TCPListDevices[BYTE_TO_INT(Crosstable[HeadAddr].NodeId)].JumpRead <= 0 THEN
					TCPListDevices[BYTE_TO_INT(Crosstable[HeadAddr].NodeId)].BlackListed:=1;
					Retry:=TRUE;
				END_IF;
			END_IF;
		END_IF;
	END_IF;
END_IF;

END_PROGRAM
